// TIA Portal V20 export
TYPE "zd_SCS_ModeBox_Outputs"
// stored: Access Published, IsFailsafeCompliant true, Namespace Safety
   STRUCT
      Disabled : Bool;   // DISABLED LT DRIVER
      PendantReq : Bool;   // PENDANT REQUIRED LT DRIVER
      Setup : Bool;   // SETUP ACTIVE
      Auto : Bool;   // AUTO READY
      Disable : Bool;   // MOTIONS DISABLED
   END_STRUCT;
END_TYPE
